TEXTLIST TextListXPIMFilters
  0 = 'Unknown'
  1 = 'T50'
  2 = 'T25'
  3 = 'T10'
  4 = 'T5'
  5 = 'T1'
  6 = 'T100'
   = ''
END_TEXTLIST

(* stored: Version 1.1.0.1, ProductVersion 3.1.4022.18
   TextList TextListXPIMFilters: Id {202aa8fc-a3e8-4e24-9efc-a37320b01e1c} *)
